{attribute 'qualified_only'}
// {attribute 'strict'}
TYPE E_StateCntrl :
(
	// Allowed to transition to Manual
	stOffline:= 0,
	// Allowed to transition to Manual/Faulted 
	stAuto:= 1,
	// Allowed to transition to Offline/Faulted/Manual 
	stManual:= 2,
	// Allowed to transition to Offline/Manual 
	stFaulted:= 3
) INT;
END_TYPE

(* stored: Version 1.1.0.1, ProductVersion 3.1.4024.4
   EnumerationTextList E_StateCntrl: Id {2d9f618a-f1f9-49a3-adc1-7e23d917bf4b} *)
